FUNCTION_BLOCK LeitungszuordnungsTester
VAR_INPUT
END_VAR
VAR_OUTPUT
END_VAR
VAR
END_VAR

IF dio.DI_1 THEN
	Visu.Ader_1:=TRUE;
ELSE 
	Visu.Ader_1 := FALSE;
END_IF

IF dio.DI_2 THEN
	Visu.Ader_2:=TRUE;
ELSE 
	Visu.Ader_2 := FALSE;
END_IF

IF dio.DI_3 THEN
	Visu.Ader_3:=TRUE;
	ELSE 
	Visu.Ader_3 := FALSE;
END_IF

IF dio.DI_4 THEN
	Visu.Ader_4:=TRUE;	
	ELSE 
	Visu.Ader_4 := FALSE;
END_IF

IF dio.DI_5 THEN
	Visu.Ader_5:=TRUE;
	ELSE 
	Visu.Ader_5 := FALSE;
END_IF

IF dio.DI_6 THEN
	Visu.Ader_6:=TRUE;
	ELSE 
	Visu.Ader_6 := FALSE;
END_IF

IF dio.DI_7 THEN
	Visu.Ader_7:=TRUE;
	ELSE 
	Visu.Ader_7 := FALSE;
END_IF

IF dio.DI_8 THEN
	Visu.Ader_8:=TRUE;
	ELSE 
	Visu.Ader_8 := FALSE;
END_IF



IF dio.DI_10 THEN
	Visu.AderErkennen:=TRUE;
	ELSE 
	Visu.AderErkennen := FALSE;
END_IF

IF dio.DI_11 THEN
	Visu.NichtVerbunden:=TRUE;
	ELSE 
	Visu.NichtVerbunden := FALSE;
END_IF

END_FUNCTION_BLOCK

(* stored: Version 1.1.0.1, ProductVersion 3.1.4022.7
   POU LeitungszuordnungsTester: Id {06128066-71dd-42f8-af82-918a0e997a69}, SpecialFunc None *)
